PROGRAM SEPARATION1
VAR
	tDelay: TON;
	bDELAY: BOOL:=FALSE;
END_VAR

tDelay(IN:=bDELAY);
CASE eSEPARATE1 OF
	E_STATION_STATE.uninit:
		eSEPARATE1:= E_STATION_STATE.idle;

	E_STATION_STATE.idle:
		bS2_RUNNING:=FALSE;
			

	E_STATION_STATE.do_action1://delay and open piston1,2
		tDELAY.PT:=T#1S;
		bDELAY:=TRUE;
		IF tDELAY.Q THEN
			bDELAY:=FALSE;
			fbPISTON[4].A_OPEN();
			fbPISTON[5].A_OPEN();
		END_IF
		
		IF fbPISTON[4].PistonStatus= ePistonStatus.OPENED  AND fbPISTON[5].PistonStatus= ePistonStatus.OPENED THEN
			eSEPARATE1:=E_STATION_STATE.do_action2;
		END_IF
		
	E_STATION_STATE.do_action2://delay and close pistons 1,2
		tDELAY.PT:=T#2S;		
		bDELAY:=TRUE;
		IF tDELAY.Q THEN
			bDELAY:=FALSE;
			fbPISTON[4].A_CLOSE();
			fbPISTON[5].A_CLOSE();
		END_IF
		IF fbPISTON[4].PistonStatus= ePistonStatus.CLOSED  AND fbPISTON[5].PistonStatus= ePistonStatus.CLOSED THEN
			eSEPARATE1:=E_STATION_STATE.do_action3;
		END_IF
	
	E_STATION_STATE.do_action3://delay
		tDELAY.PT:=T#2S;
		bDELAY:=TRUE;
		IF tDELAY.Q THEN
			bDELAY:=FALSE;
			eSEPARATE1:=E_STATION_STATE.done;
		END_IF
		
	
	E_STATION_STATE.done:
		bS2_RUNNING:=FALSE;
		
	E_STATION_STATE.pause:
		//paused

END_CASE

END_PROGRAM

(* stored: Version 1.1.0.1, ProductVersion 3.1.4024.12
   POU SEPARATION1: Id {0a3315b2-61c0-4450-961e-215e0d8b923c}, SpecialFunc None *)
